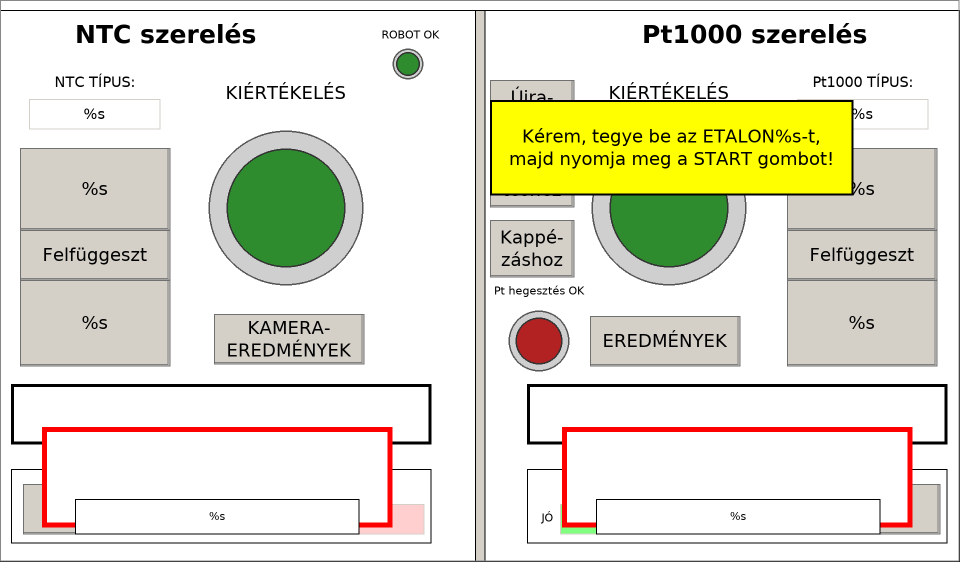
VISUALIZATION Termeles0  // 960x562
    Rectangle (0,10 960x552)
    RoundedRectangle (11,384 420x60), tooltip "Állapotváltozó: %s", text list: 'AUTOMATA_lepesek1', text index: AUTOMATA.iState
        p4168582468: AUTOMATA.iState
    Group (527,469 420x74)
        Rectangle (0,0 420x74)
        Textfield (33,35 81x30), "%s", text variable: GVL.nGoodProductCount
        Label (8,34 25x30), "JÓ"
        Textfield (170,35 81x30), "%s", text variable: GVL.nBadProductCount
        Label (128,34 42x30), "HIBÁS"
        Label (103,0 82x30), "DARABSZÁM"
        Button (263,15 150x50), "NULLÁZ"
            OnMouseUp: execute { GVL.nGoodProductCount:=0; GVL.nBadProductCount:=0; }
    RoundedRectangle (527,384 420x60), tooltip "Állapotváltozó: %s", text list: 'AUTOMATA_lepesek2', text index: AUTOMATA.iState2
        p4168582468: AUTOMATA.iState2
    Label (645,19 220x30), "Pt1000 szerelés"
    Group (579,78 180x220)
        Lamp1 (0,40 180x180), variable: GVL.bProductNOK, style: Lamp-Lamp1-Red
        Lamp1 (0,40 180x180), variable: GVL.bProductOK, invisible if: GVL.bProductNOK, style: Lamp-Lamp1-Green
        Label (0,0 180x30), "KIÉRTÉKELÉS"
    Button (787,148 150x82), "%s", text variable: AUTOMATA.sStart2GombFelirat, colour toggle: GVL.nElectrode3Usage>GVL.nElectrode3UsageWarn, input disabled if: NOT (ABS(PISTITENGELY.lrPistiActPos-GVL.lrPtSzervizbox)<0.1) AND NOT AUTOMATA.bContinue2En
        p573394764: GVL.nElectrode3AlarmColor
        OnMouseUp: execute {
            IF AUTOMATA.iState2=0 THEN
            	AUTOMATA.iState2:=1;
            ELSE
            	AUTOMATA.bContinue2:=TRUE;
            END_IF
        }
    Button (787,280 150x86), "%s", text variable: AUTOMATA.sStop2GombFelirat, input disabled if: (AUTOMATA.iState2=0) AND ABS(PISTITENGELY.lrPistiActPos-GVL.lrPtSzervizbox)<0.1
        OnMouseUp: execute {
            IF NOT(AUTOMATA.iState2=99) THEN
            //	AUTOMATA.bContinue2:=FALSE;
            //	AUTOMATA.bWelderReservedBy2:=FALSE;
            //	AUTOMATA.bRobotReservedBy2:=FALSE;
            //	GVL.bAdapterLefogo:=FALSE;
            //	AUTOMATA.sStop2GombFelirat:='Szervízboxhoz';
            //	AUTOMATA.bStart2GombTiltva:=TRUE;
            //	AUTOMATA.sStart2GombFelirat:='START';
            //	PISTITENGELY.sPistiAxisCommand:='STOP';
            //	AUTOMATA.iState2:=0;
            	AUTOMATA.iState2:=200;
            ELSE
            	AUTOMATA.iState2:=100;
            END_IF
        }
    Button (590,316 150x50), "EREDMÉNYEK"
        OnMouseUp: execute { GVL.bMeresiEredmenyekRejtve:=FALSE; }
    Group (11,469 420x74)
        Rectangle (0,0 420x74)
        Textfield (195,35 81x30), "%s", text variable: GVL.nGoodProductCount1
        Label (170,34 25x30), "JÓ"
        Textfield (332,35 81x30), "%s", text variable: GVL.nBadProductCount1
        Label (290,34 42x30), "HIBÁS"
        Label (265,0 82x30), "DARABSZÁM"
        Button (12,15 150x50), "NULLÁZ"
            OnMouseUp: execute { GVL.nGoodProductCount1:=0; GVL.nBadProductCount1:=0; }
    Button (20,148 150x82), "%s", text variable: AUTOMATA.sStart1GombFelirat, colour toggle: (GVL.nElectrode1Usage>GVL.nElectrode1UsageWarn) OR (GVL.nElectrode2Usage>GVL.nElectrode2UsageWarn), input disabled if: AUTOMATA.bStart1GombTiltva
        p573394764: MIN(GVL.nElectrode1AlarmColor,GVL.nElectrode2AlarmColor)
        OnMouseUp: execute {
            IF AUTOMATA.iState=0 THEN
            	AUTOMATA.iState:=1;
            ELSE
            	AUTOMATA.bContinue:=TRUE;
            END_IF
        }
    Button (20,280 150x86), "%s", text variable: AUTOMATA.sStop1GombFelirat, input disabled if: (AUTOMATA.iState=0) AND ABS(JOZSITENGELY.lrJozsiActPos-GVL.lrNTCSzervizbox)<0.1
        OnMouseUp: execute {
            AUTOMATA.bStopMegnyomva:=TRUE;
            //IF NOT(AUTOMATA.iState=0) THEN
            //	AUTOMATA.bContinue:=FALSE;
            //	AUTOMATA.bWelderReservedBy1:=FALSE;
            //	AUTOMATA.bRobotReservedBy1:=FALSE;
            //	JOZSITENGELY.sJozsiAxisCommand:='STOP';
            //	AUTOMATA.iState:=0;
            //	AUTOMATA.iState:=130;
            //ELSE
            //	AUTOMATA.iState:=100;
            //END_IF
        }
    Label (66,19 200x30), "NTC szerelés"
    Group (196,78 180x220)
        Lamp1 (0,40 180x180), variable: GVL.bProduct1NOK, style: Lamp-Lamp1-Red
        Lamp1 (0,40 180x180), variable: GVL.bProduct1OK, invisible if: GVL.bProduct1NOK, style: Lamp-Lamp1-Green
        Label (0,0 180x30), "KIÉRTÉKELÉS"
    Rectangle (475,10 10x552)
    Label (40,67 110x30), "NTC TÍPUS:"
    Textfield (29,99 131x30), "%s", text variable: GVL.sNTCTypeElozo, colour toggle: GVL.sNTCType='HIBÁS KÓD'
        OnMouseClick: write GVL.sNTCType via Edit
    Label (808,67 110x30), "Pt1000 TÍPUS:"
    Textfield (797,99 131x30), "%s", text variable: GVL.sPtTypeElozo, colour toggle: GVL.sPtType='HIBÁS KÓD'
        OnMouseClick: write GVL.sPtType via Edit
    Button (490,80 84x57), "Újra- mérés", text variable: AUTOMATA.sStart2GombFelirat, colour toggle: AUTOMATA.bUjrameres, pressed state: AUTOMATA.bUjrameres, invisible if: TRUE
        OnMouseClick: execute {
            AUTOMATA.bUjrameres:=NOT AUTOMATA.bUjrameres;
            IF AUTOMATA.bUjrameres THEN
            	AUTOMATA.bHegesztes6Be:=GVL.bHegesztes6Be;
            	AUTOMATA.bHegesztes7Be := GVL.bHegesztes7Be;
            	AUTOMATA.bPtKameraBe := GVL.bPtKameraBe;
            	AUTOMATA.bRobotKappeBe := GVL.bRobotKappeBe;
            	AUTOMATA.bKappeBe := GVL.bKappeBe;
            	AUTOMATA.bMeresBe := GVL.bMeresBe;
            	AUTOMATA.bJelolesBe := GVL.bJelolesBe;
            	GVL.bHegesztes6Be := FALSE;
            	GVL.bHegesztes7Be := FALSE;
            	GVL.bPtKameraBe := FALSE;
            	GVL.bRobotKappeBe := FALSE;
            	GVL.bKappeBe := TRUE;
            	GVL.bMeresBe := TRUE;
            	GVL.bJelolesBe := TRUE;
            ELSE
            	GVL.bHegesztes6Be:=AUTOMATA.bHegesztes6Be;
            	GVL.bHegesztes7Be := AUTOMATA.bHegesztes7Be;
            	GVL.bPtKameraBe := AUTOMATA.bPtKameraBe;
            	GVL.bRobotKappeBe := AUTOMATA.bRobotKappeBe;
            	GVL.bKappeBe := AUTOMATA.bKappeBe;
            	GVL.bMeresBe := AUTOMATA.bMeresBe;
            	GVL.bJelolesBe := AUTOMATA.bJelolesBe;
            END_IF
        }
    Button (787,230 150x50), "Felfüggeszt", pressed state: AUTOMATA.bFelfuggeszt2
        OnMouseUp: execute {
            IF AUTOMATA.bFelfuggeszt2=FALSE THEN
            	AUTOMATA.bFelfuggeszt2:=TRUE;
            	AUTOMATA.iState2Elozo:=AUTOMATA.iState2;
            	AUTOMATA.iState2:=300;
            ELSE
            	AUTOMATA.bFelfuggeszt2:=FALSE;
            END_IF
        }
    Button (20,230 150x50), "Felfüggeszt", pressed state: AUTOMATA.bFelfuggeszt
        OnMouseUp: execute {
            IF AUTOMATA.bFelfuggeszt=FALSE THEN
            	AUTOMATA.bFelfuggeszt:=TRUE;
            	AUTOMATA.iStateElozo:=AUTOMATA.iState;
            	AUTOMATA.iState:=300;
            ELSE
            	AUTOMATA.bFelfuggeszt:=FALSE;
            END_IF
        }
    Group (42,427 350x107)
        RoundedRectangle (0,0 350x100), invisible if: GVL.bHibauzenetNTCRejtve, text list: 'ErrorList', text index: GVL.nHibaKodNTC
        Rectangle (33,72 284x35), "%s", text variable: AUTOMATA.sRobotHiba, invisible if: GVL.bHibauzenetNTCRejtve OR NOT (GVL.nHibaKodNTC=307)
    Group (562,427 350x107)
        RoundedRectangle (0,0 350x100), invisible if: GVL.bHibauzenetPtRejtve, text list: 'ErrorList', text index: GVL.nHibaKodPt
        Rectangle (34,72 284x35), "%s", text variable: AUTOMATA.sRobotHiba, invisible if: GVL.bHibauzenetPtRejtve OR NOT (GVL.nHibaKodPt=307)
    Button (214,314 150x50), "KAMERA- EREDMÉNYEK"
        OnMouseUp: execute {
            GVL.bNTCBezarGombRejtve:=FALSE;
            GVL.bKameraEredmenyekRejtve:=FALSE;
            GVL.iBitmap_Version:=GVL.iBitmap_Version+1;
        }
    Group (486,281 106x95), invisible if: TRUE
        Label (0,0 106x20), "Pt hegesztés OK"
        Lamp1 (18,25 70x70), variable: GVL.bPtKameraHegesztesOK, style: Lamp-Lamp1-Green
        Lamp1 (18,25 70x70), variable: NOT GVL.bPtKameraHegesztesOK, invisible if: GVL.bPtKameraTrigger OR GVL.bPtKameraHegesztesOK OR AUTOMATA.bPtKameraHasznalatlan, style: Lamp-Lamp1-Red
    Button (490,150 84x57), "Hegesz- téshez", invisible if: (GVL.bPtKameraBe=TRUE) AND (AUTOMATA.bPtKameraGombokEnged=FALSE)
        tap AUTOMATA.bHegeszteshezGomb
    Button (490,220 84x57), "Kappé- záshoz", invisible if: (GVL.bPtKameraBe=TRUE) AND (AUTOMATA.bPtKameraGombokEnged=FALSE)
        tap AUTOMATA.bKappezashozGomb
    RoundedRectangle (490,100 363x95), "Kérem, tegye be az ETALON%s-t, majd nyomja meg a START gombot!", text variable: GVL.iCurrentProductType+4, invisible if: NOT (GVL.iCurrentProductType<0) OR NOT GVL.bMeresBe
    Label (360,20 101x30), "ROBOT OK", invisible if: ROBOTREMOTE.bRobotCommOpen=FALSE
    Lamp1 (390,46 36x36), variable: RobotProcess.baStatus[9], invisible if: ROBOTREMOTE.bRobotCommOpen=FALSE, style: Lamp-Lamp1-Green
END_VISUALIZATION

(* stored: Version 1.1.0.1, ProductVersion 3.1.4024.11
   Visu Termeles0: Id {50c48183-5e17-49bb-8d14-651d4ecfe0e5} *)
